TYPE ST_FeedbackQualisys :
STRUCT
	dist: LREAL;
	pos: ARRAY[0..2] OF LREAL;
END_STRUCT
END_TYPE

(* stored: Version 1.1.0.1, ProductVersion 3.1.4026.8
   DUT ST_FeedbackQualisys: Id {24549d75-2338-4db0-b4b2-661ae5b5c927} *)
